Fanuc KAREL source: CLR_POS_REG.kl

PROGRAM T
%NOLOCKGROUP
VAR
 v0 : INTEGER
 v1 : INTEGER
 v2 : INTEGER
BEGIN
 CLR_POS_REG(v0, v1, v2)
END T
